Yaskawa INFORM job: SPOT_WELD.JBI

/JOB
//NAME SPOT_WELD
//POS
///NPOS 0,0,0,0,0,0
//INST
///DATE 2022/06/13 02:25
///ATTR SC,RW,MC
///LVARS 5,0,5,0,0,0,0,0
NOP
'GUARDA ARGUMENTO 1
'(IDENTIFICACAO PONTO DE SOLDA)
GETARG LB000 IARG#(1)
'
'GUARDA ARGUMENTO 2
'NUMERO BYTE COM ID PONTO SOLDA
GETARG LD000 IARG#(2)
'
'MOVE PARA VARIAVEL VALOR DECIMAL
'SETADO NO BYTE DE INPUT COM
'NUMERO DO PROGRAMA PARA AJUSTE
'DO PONTO DE SOLDA
DIN LB001 IG#(LD000)
'
IFTHENEXP LB000=LB001
	'
	 PULSE OT#(2912) T=1.00
	'
ENDIF
'
END
